                               IF (#statDeviceFaultyModules[#tempSlotIndex + 1] = TRUE)
                               THEN
                                   // Fault in module
                                   #ioSystemData.devices[#tempDeviceIndex].slots[#tempSlotIndex].faulty := TRUE;
                                   #ioSystemData.devices[#tempDeviceIndex].slots[#tempSlotIndex].state := #STATE_FAULT;
                               END_IF;
                           ELSE
                               #ioSystemData.devices[#tempDeviceIndex].slots[#tempSlotIndex].error := FALSE;
                               #ioSystemData.devices[#tempDeviceIndex].slots[#tempSlotIndex].problem := FALSE;
                               #ioSystemData.devices[#tempDeviceIndex].slots[#tempSlotIndex].faulty := FALSE;
                           END_IF;

                           IF (#statDeviceExistingModules[#tempSlotIndex + 1] = TRUE)
                           THEN
                               // Module exists
                               #ioSystemData.devices[#tempDeviceIndex].slots[#tempSlotIndex].exists := TRUE;
                           ELSE
                               // Module does not exist
                               #ioSystemData.devices[#tempDeviceIndex].slots[#tempSlotIndex].exists := FALSE;
                           END_IF;
                       END_IF;
                   END_FOR;
               ELSE
                   // All modules are okay
                   FOR #tempSlotIndex := 0 TO "USERDIAG_SLOTS_PER_DEVICE_UPPER_LIM" DO
                       IF (#ioSystemData.devices[#tempDeviceIndex].slots[#tempSlotIndex].configured = TRUE)
                       THEN
                           #ioSystemData.devices[#tempDeviceIndex].slots[#tempSlotIndex].error := FALSE;
                           #ioSystemData.devices[#tempDeviceIndex].slots[#tempSlotIndex].problem := FALSE;
                           #ioSystemData.devices[#tempDeviceIndex].slots[#tempSlotIndex].faulty := FALSE;
                           #ioSystemData.devices[#tempDeviceIndex].slots[#tempSlotIndex].exists := TRUE;
                       END_IF;
                   END_FOR;
           END_CASE;
       END_IF;

       // Initialize the pointer for the next run
       #tempDeviceIndex := #ioSystemData.devices[#tempDeviceIndex].nextDevice;
   END_WHILE;


   // Write static values to outputs
   #error := #statError;
   #status := #statStatus;
   #statusID := #statStatusID;
END_FUNCTION_BLOCK

FUNCTION_BLOCK "HMI: Network Health"   // FB31, SCL
{ S7_Optimized_Access := 'TRUE' }
VERSION : 0.1
   VAR_IN_OUT
      ioSystemData : Array[1.."USERDIAG_IO_SYSTEMS_UPPER_LIM"] of "UserDiag_typeIOSystem";
      netHealthScreen : "Network Health Screen";
   END_VAR
   VAR_TEMP
      i : Int;
      animate : Struct
         ok : USInt;
         faulty : USInt;
         lostConn : USInt;
         disabled : USInt;
         problem : USInt;
         wasFaulty : USInt;
         wasLost : USInt;
         wasDisabled : USInt;
         problemGone : USInt;
      END_STRUCT;
   END_VAR
   VAR CONSTANT
      statOk : USInt := 1;
   END_VAR
BEGIN
   #animate.ok := "BgDGr";

   FOR #i := 1 TO "pnioDeviceCount" DO
       #netHealthScreen.pnioDevices[#i].label := #ioSystemData[1].devices[#i].name;
       CASE #ioSystemData[1].devices[#i].state OF
           #statOk:
               #netHealthScreen.pnioDevices[#i].animate := #animate.ok;
           ELSE 
               ;
       END_CASE;
   END_FOR;
END_FUNCTION_BLOCK

FUNCTION_BLOCK "HSS: Driver"   // FB32, LAD
{ S7_Optimized_Access := 'TRUE' }
VERSION : 0.1
   VAR_INPUT
      mLs : "Recipe: Libraries";
   END_VAR
   VAR_IN_OUT
      stations : "Stations";
      hmis : Array[0.."hmiStnCount"] of "HSS: Compressed";
   END_VAR
   VAR
      recipeSelector : Array[0.."hmiStnCount"] of Int;
      r1 : Array[0.."hmiStnCount"] of DInt;
      instsHSSMenuSelect : Array[0.."hmiStnCount"] of "HSS: Recipe Selection";
      instsHSSPartSelect : Array[0.."hmiStnCount"] of "HSS: Part Selection";
   END_VAR
   VAR_TEMP
      i : Int;
   END_VAR
   VAR CONSTANT
      hssOffset : Int := 25;
   END_VAR
BEGIN

REGION Network 1 (SCL): TEMPLATE SCREENS
   FOR #i := 0 TO "hmiStnCount" DO
       "HSS: Template"(menuLibrary := #mLs.stations[#i + #hssOffset],
                       menuSelector := #recipeSelector[#i],
                       tmplt := #hmis[#i].scrnTmplt);
       #instsHSSMenuSelect[#i](lib := #mLs.stations[#i + #hssOffset],
                               slctScreen := #hmis[#i].scrnSlctMn,
                               r1 := #r1[#i],
                               station := #stations.me[#i + #hssOffset],
                               recipeSelector := #recipeSelector[#i]);
       #instsHSSPartSelect[#i](recipeNum:= #recipeSelector[#i],
                              lib:=#mLs.stations[#i + #hssOffset],
                              slctScreen:=#hmis[#i].scrnSlctPrt,
                              station:=#stations.me[#i + #hssOffset]);

   END_FOR;
END_REGION
END_FUNCTION_BLOCK

FUNCTION_BLOCK "HSS: Part Selection"   // FB33, SCL
{ S7_Optimized_Access := 'TRUE' }
VERSION : 0.1
   VAR_INPUT
      recipeNum : Int;
      lib : "Recipe: Library";
   END_VAR
   VAR_IN_OUT
      slctScreen : "HSS: Part Selection Screen";
      station : "Station";
   END_VAR
   VAR
      oldBtnsIn : Array[0..31] of Bool;
   END_VAR
   VAR_TEMP
      eval : "HSS: Part Selection Screen";
      i : Int;
      btnsIn : Array[0..31] of Bool;
      btnStates : Array[0.."ptsPerStn"] of Bool;
   END_VAR
BEGIN
   #eval := #slctScreen;


   SCATTER(IN := #slctScreen.pbs ,
           OUT => #btnsIn);
   #btnStates := #station.btnStates;


   FOR #i := 0 TO "ptsPerStn" DO
       IF #btnsIn[#i] AND #btnsIn[#i] <> #oldBtnsIn[#i] THEN
           #btnStates[#i] := NOT #btnStates[#i];
       END_IF;
   END_FOR;


   FOR #i := 0 TO "ptsPerStn" DO
       "Part Select Button"(recipeNum := #recipeNum,
                            lib := #lib,
                            actuate := #btnsIn[#i],
                            btnNum := #i,
                            stn:= #station,
                            partSelectScreen := #eval);
   END_FOR;


   #station.btnStates := #btnStates;
   #oldBtnsIn := #btnsIn;
   #slctScreen := #eval;
END_FUNCTION_BLOCK

FUNCTION_BLOCK "Table Navigatio"   // FB34, SCL
{ S7_Optimized_Access := 'TRUE' }
VERSION : 0.1
   VAR_INPUT
      maxRows : DInt;
      visRows : DInt;
      offset : DInt;
      trigger : Bool;
   END_VAR
   VAR_IN_OUT
      r1 : DInt;
      rowIndices : Array[0..#maxOutRows] of DInt;
   END_VAR
   VAR
      old : Struct
         trigger : Bool := false;
      END_STRUCT;
   END_VAR
   VAR_TEMP
      i : DInt;
      output : Array[0..#maxOutRows] of DInt;
      thisIndex : DInt;
      newR1 : DInt;
   END_VAR
   VAR CONSTANT
      maxOutRows : DInt := 99;
   END_VAR
BEGIN
   IF #trigger AND NOT #old.trigger THEN

       FOR #i := 0 TO #maxOutRows DO
           #output[#i] := -1;
       END_FOR;

       IF #offset > -1000 THEN

           #newR1 := #r1 + #offset;

           IF #newR1 < 0 THEN
               #newR1 := #newR1 + #maxRows;
           END_IF;

           IF #newR1 > #maxRows THEN
               #newR1 := #newR1 - #maxRows;
           END_IF;

       END_IF;

       IF #offset = -1000 THEN
           #newR1 := 0;
       END_IF;

       IF #offset = - 2000 THEN
           #newR1 := #maxRows - #visRows;
       END_IF;

       FOR #i := 0 TO #visRows - 1 DO
           #thisIndex := #newR1 + #i;
           IF #thisIndex < 0 THEN
               #thisIndex := #thisIndex + #maxRows;
           END_IF;
           IF #thisIndex >= #maxRows THEN
               #thisIndex := #thisIndex - #maxRows;
           END_IF;
           #output[#i] := #thisIndex;
       END_FOR;

       #rowIndices := #output;
       #r1 := #newR1;

   END_IF;

   #old.trigger := #trigger;
END_FUNCTION_BLOCK

FUNCTION_BLOCK "HSS: Recipe Selection"   // FB35, SCL
{ S7_Optimized_Access := 'TRUE' }
VERSION : 0.1
   VAR_INPUT
      lib : "Recipe: Library";
   END_VAR
   VAR_IN_OUT
      slctScreen : "HSS: Menu Selection Screen";
      r1 : DInt;
      recipeSelector : Int;
      station : "Station";
   END_VAR
   VAR
      old : Struct
         navPress : Bool;
      END_STRUCT;
      instTableNavigation : "Table Navigatio";
   END_VAR
   VAR_TEMP
      eval : "HSS: Menu Selection Screen";
      pbs : Array[0..#pbFlagCnt] of Bool;
      POS : DInt;
      status : DInt;
      i : Int;
      btnNum : Int;
      pRowVisLbl : Int;
      pRowInvisLbl : Int;
      pRecipeInvisLbl : Int;
      pRecipeVisLbl : Int;
      pRecipeLib : Int;
      pRowTxt : Int;
      pRecipeTxt : Int;
      shifter : DWord;
      btnsAsBool : Array[0..31] of Bool;
      rows : Array[0..99] of DInt;
      offset : DInt;
      navPress : Bool;
      selPress : Bool;
      maxRows : DInt;
      tmrReal : Real;
      partNumber : WString;
   END_VAR
   VAR CONSTANT
      pbFlagCnt : Int := 31;
      btnCnt : Int := 5;
      navMask : DWord := 16#0000_003F;
      visRows : DInt := 6;
      home : DInt := -1000;
      end : DInt := -2000;
      alotted : Real := 1800.0;
      critical : Real := 300.0;
   END_VAR
BEGIN
   REGION "INITITALIZE LOCALS"
       #eval := #slctScreen;
       #maxRows := #lib.size;
       SCATTER(IN := #eval.pbs,
               OUT => #btnsAsBool);
   END_REGION


   REGION "GET RECIPE SELECTION PRESS" 
       FOR #i := 6 TO 31 DO
           IF #btnsAsBool[#i] THEN
               #recipeSelector := DINT_TO_INT(#r1) + #i - 6;
               #selPress := TRUE;
               EXIT;
           END_IF;
       END_FOR;
       FOR #i := 0 TO "ptsPerStn" DO
           #station.partNumbers[#i] := #lib.raw[#recipeSelector, #i];
           // IF #i = 1 THEN
           //     #station.partNumbers[#i] := WSTRING#'';
           // END_IF;

       END_FOR;
       REGION "LOOP THROUGH BUTTONS"
           FOR #i := 0 TO "ptsPerStn" DO

               REGION "COPY TO LOCAL"
                   #partNumber := #station.partNumbers[#i];
               END_REGION

               REGION "IF BUTTON HAS ASSOCIATED PN"
                   IF LEN(#partNumber) <> 0 THEN

                       REGION "COPY TO LOCAL"
                           #tmrReal := #station.presetTime.allotted[#i];
                       END_REGION

                       REGION "ON NO TIME ENTERED"
                           IF #tmrReal = 0.0 THEN

                               REGION "ASSIGN ALLOTTED VALUES"
                                   #station.presetTime.allotted[#i] := #alotted;
                               END_REGION

                           END_IF;
                       END_REGION

                       REGION "COPY TO LOCAL"
                           #tmrReal := #station.presetTime.critical[#i];
                       END_REGION

                       REGION "ON NO TIME ENTERED"
                           IF #tmrReal = 0.0 THEN

                               REGION "ASSIGN CRITICAL VALUES"
                                   #station.presetTime.critical[#i] := #critical;
                               END_REGION

                           END_IF;
                       END_REGION

                   END_IF;
               END_REGION

               REGION "IF BUTTON HAS NO ASSOCIATED PN"
                   IF LEN(#partNumber) = 0 THEN

                       REGION "COPY TO LOCAL"
                           #tmrReal := #station.presetTime.allotted[#i];
                       END_REGION

                       REGION "ON NO TIME ENTERED"
                           IF #tmrReal <> 0.0 THEN

                               REGION "ASSIGN ALLOTTED VALUES"
                                   #station.presetTime.allotted[#i] := 0.0;
                               END_REGION

                           END_IF;
                       END_REGION

                       REGION "COPY TO LOCAL"
                           #tmrReal := #station.presetTime.critical[#i];
                       END_REGION

                       REGION "ON NO TIME ENTERED"
                           IF #tmrReal <> 0.0 THEN

                               REGION "ASSIGN CRITICAL VALUES"
                                   #station.presetTime.critical[#i] := 0.0;
                               END_REGION

                           END_IF;
                       END_REGION

                   END_IF;
               END_REGION


           END_FOR;
       END_REGION
   END_REGION


   REGION "TABLE NAVIGATION"
       IF #maxRows > #visRows THEN
           IF #eval.pbs.%X0 THEN
               #offset := #home;
           END_IF;
           IF #eval.pbs.%X1 THEN
               #offset := -1 * #visRows;
           END_IF;
           IF #eval.pbs.%X2 THEN
               #offset := -1;
           END_IF;
           IF #eval.pbs.%X3 THEN
               #offset := 1;
           END_IF;
           IF #eval.pbs.%X4 THEN
               #offset := #visRows;
           END_IF;
           IF #eval.pbs.%X5 THEN
               #offset := #end;
           END_IF;

           IF (#eval.pbs AND #navMask) <> 0 THEN
               #navPress := true;
           END_IF;

           #instTableNavigation(maxRows := #maxRows,
                                visRows := #visRows,
                                offset := #offset,
                                trigger := #navPress,
                                r1 := #r1,
                                rowIndices := #rows);
       END_IF;

       IF #maxRows <= #visRows THEN
           FOR #i := 0 TO #visRows - 1 DO
               #rows[#i] := #i;
           END_FOR;
       END_IF;

   END_REGION


   REGION "CA: NAV BUTTONS"
       FOR #i := 0 TO #visRows - 1 DO
           "Recipe Nav Button"(visRows := DINT_TO_INT(#visRows),
                               actuate := #btnsAsBool[#i],
                               maxRows := DINT_TO_INT(#maxRows),
                               btnNum := #i,
                               recipeSelectScreen := #eval);
       END_FOR;
   END_REGION



   REGION "ODA: RECIPE SELECT BUTTONS"
       IF (#navPress AND NOT #old.navPress) OR
           (#maxRows <= #visRows) THEN

           FOR #i := 0 TO #visRows - 1 DO
               "Recipe Select Button"(visRows := DINT_TO_INT(#visRows),
                                      rowNum := DINT_TO_INT(#rows[#i]),
                                      lib := #lib,
                                      actuate := #btnsAsBool[#i + 6],
                                      maxRows := DINT_TO_INT(#maxRows),
                                      btnNum := #i,
                                      recipeSelectScreen := #eval);
           END_FOR;

       END_IF;
   END_REGION


   REGION "CHANGE DETECTION"
       #old.navPress := #navPress;
   END_REGION


   REGION "COPY TO GLOBAL"
       #slctScreen := #eval;
   END_REGION
END_FUNCTION_BLOCK

FUNCTION_BLOCK "KP8 Driver"   // FB101, SCL
{ S7_Optimized_Access := 'FALSE' }
VERSION : 0.1
   VAR_INPUT
      btnIn : Byte;   // byte that contains input data from kp8 buttons
      hardInit : Bool;   // initializes function. can be used for reset
      softInit : Bool;
      btn0Activate : Bool;   // true for on, false for off
      btn0Mode : Bool;   // true for maintained, false for momentary
      btn0Group : Int;
      btn0Flash : Bool;
      btn0ColorOn1 : String[10];   // enter: red OR green OR blue OR yellow OR white OR off
      btn0ColorOn2 : String[10];
      btn0ColorOff : String[10];   // enter: red OR green OR blue OR yellow OR white OR off
      btn1Activate : Bool;   // true for on, false for off
      btn1Mode : Bool;   // true for maintained, false for momentary
      btn1Group : Int;
      btn1Flash : Bool;
      btn1ColorOn1 : String[10];   // enter: red OR green OR blue OR yellow OR white OR off
      btn1ColorOn2 : String[10];
      btn1ColorOff : String[10];   // enter: red OR green OR blue OR yellow OR white OR off
      btn2Activate : Bool;   // true for on, false for off
      btn2Mode : Bool;   // true for maintained, false for momentary
      btn2Group : Int;
      btn2Flash : Bool;
      btn2ColorOn1 : String[10] := '';   // enter: red OR green OR blue OR yellow OR white OR off
      btn2ColorOn2 : String[10];
      btn2ColorOff : String[10];   // enter: red OR green OR blue OR yellow OR white OR off
      btn3Activate : Bool;   // true for on, false for off
      btn3Mode : Bool;   // true for maintained, false for momentary
      btn3Group : Int;
      btn3Flash : Bool;
      btn3ColorOn1 : String[10];   // enter: red OR green OR blue OR yellow OR white OR off
      btn3ColorOn2 : String[10];
      btn3ColorOff : String[10];   // enter: red OR green OR blue OR yellow OR white OR off
      btn4Activate : Bool;   // true for on, false for off
      btn4Mode : Bool;   // true for maintained, false for momentary
      btn4Group : Int;
      btn4Flash : Bool;
      btn4ColorOn1 : String[10];   // enter: red OR green OR blue OR yellow OR white OR off
      btn4ColorOn2 : String[10];
      btn4ColorOff : String[10];   // enter: red OR green OR blue OR yellow OR white OR off
      btn5Activate : Bool;   // true for on, false for off
      btn5Mode : Bool;   // true for maintained, false for momentary
      btn5Group : Int;
      btn5Flash : Bool;
      btn5ColorOn1 : String[10];   // enter: red OR green OR blue OR yellow OR white OR off
      btn5ColorOn2 : String[10];
      btn5ColorOff : String[10];   // enter: red OR green OR blue OR yellow OR white OR off
      btn6Activate : Bool;   // true for on, false for off
      btn6Mode : Bool;   // true for maintained, false for momentary
      btn6Group : Int;
      btn6Flash : Bool;
      btn6ColorOn1 : String[10];   // enter: red OR green OR blue OR yellow OR white OR off
      btn6ColorOn2 : String[10];
      btn6ColorOff : String[10];   // enter: red OR green OR blue OR yellow OR white OR off
      btn7Activate : Bool;   // true for on, false for off
      btn7Mode : Bool;   // true for maintained, false for momentary
      btn7Group : Int;
      btn7Flash : Bool;
      btn7ColorOn1 : String[10];   // enter: red OR green OR blue OR yellow OR white OR off
      btn7ColorOn2 : String[10];
      btn7ColorOff : String[10];   // enter: red OR green OR blue OR yellow OR white OR off
   END_VAR
   VAR_OUTPUT
      btnStatesOut : Array[0..7] of Bool;   // the output array represents the state of button presses
      btnColorsOut : DWord;
   END_VAR
   VAR
      mask : Byte;
      btnInInt : Byte;
      btnEval : Byte;
      i1 : Int;
      i2 : Int;
      btnActivateInt : Array[0..7] of Bool;
      btnClrMskOffInt : Array[0..7] of DWord;
      btnClrMskOn1Int : Array[0..7] of DWord;
      btnClrMskOn2Int : Array[0..7] of DWord;
      btnClrOffInt : Array[0..7] of String[10];
      btnClrOn1Int : Array[0..7] of String[10];
      btnClrOn2Int : Array[0..7] of String[10];
      btnColors : DWord;
      btnInArrayNew : Array[0..7] of Bool;
      btnInArrayOld : Array[0..7] of Bool;
      btnStateArrayInt : Array[0..7] of Bool;
      btnModeInt : Array[0..7] of Bool;
      btnFlashInt : Array[0..7] of Bool;
      btnGroup : Array[0..7] of Int;
   END_VAR
   VAR CONSTANT
      btnMskRed : DWord := dw#16#0100_0000;
      btnMskGreen : DWord := dw#16#0001_0000;
      btnMskBlue : DWord := dw#16#000_0100;
      btnMskYellow : DWord := dw#16#0101_0000;
      btnMskWhite : DWord := dw#16#0101_0100;
      btnMskBlack : DWord := dw#16#FEFE_FEFF;
      initBtnColors : DWord := dw#16#0000_0000;
   END_VAR
BEGIN
   REGION "ALL INITS"
       IF #hardInit OR #softInit THEN

           REGION "CLEAR OUTPUT COLORS"
               #btnColors := #initBtnColors;
           END_REGION

           REGION "TRANSFER PARAMETERS TO INTERNAL ARRAYS"

               REGION "BUTTON 0"
                   #btnActivateInt[0] := #btn0Activate;
                   #btnModeInt[0] := #btn0Mode;
                   #btnGroup[0] := #btn0Group;
                   #btnClrOn1Int[0] := #btn0ColorOn1;
                   #btnClrOn2Int[0] := #btn0ColorOn2;
                   #btnClrOffInt[0] := #btn0ColorOff;
               END_REGION

               REGION "BUTTON 1"
                   #btnActivateInt[1] := #btn1Activate;
                   #btnModeInt[1] := #btn1Mode;
                   #btnGroup[1] := #btn1Group;
                   #btnClrOn1Int[1] := #btn1ColorOn1;
                   #btnClrOn2Int[1] := #btn1ColorOn2;
                   #btnClrOffInt[1] := #btn1ColorOff;
               END_REGION

               REGION "BUTTON 2"
                   #btnActivateInt[2] := #btn2Activate;
                   #btnModeInt[2] := #btn2Mode;
                   #btnGroup[2] := #btn2Group;
                   #btnClrOn1Int[2] := #btn2ColorOn1;
                   #btnClrOn2Int[2] := #btn2ColorOn2;
                   #btnClrOffInt[2] := #btn2ColorOff;
               END_REGION

               REGION "BUTTON 3"
                   #btnActivateInt[3] := #btn3Activate;
                   #btnModeInt[3] := #btn3Mode;
                   #btnGroup[3] := #btn3Group;
                   #btnClrOn1Int[3] := #btn3ColorOn1;
                   #btnClrOn2Int[3] := #btn3ColorOn2;
                   #btnClrOffInt[3] := #btn3ColorOff;
               END_REGION

               REGION "BUTTON 4"
                   #btnActivateInt[4] := #btn4Activate;
                   #btnModeInt[4] := #btn4Mode;
                   #btnGroup[4] := #btn4Group;
                   #btnClrOn1Int[4] := #btn4ColorOn1;
                   #btnClrOn2Int[4] := #btn4ColorOn2;
                   #btnClrOffInt[4] := #btn4ColorOff;
               END_REGION

               REGION "BUTTON 5"
                   #btnActivateInt[5] := #btn5Activate;
                   #btnModeInt[5] := #btn5Mode;
                   #btnGroup[5] := #btn5Group;
                   #btnClrOn1Int[5] := #btn5ColorOn1;
                   #btnClrOn2Int[5] := #btn5ColorOn2;
                   #btnClrOffInt[5] := #btn5ColorOff;
               END_REGION

               REGION "BUTTON 6"
                   #btnActivateInt[6] := #btn6Activate;
                   #btnModeInt[6] := #btn6Mode;
                   #btnGroup[6] := #btn6Group;
                   #btnClrOn1Int[6] := #btn6ColorOn1;
                   #btnClrOn2Int[6] := #btn6ColorOn2;
                   #btnClrOffInt[6] := #btn6ColorOff;
               END_REGION

               REGION "BUTTON 7"
                   #btnActivateInt[7] := #btn7Activate;
                   #btnModeInt[7] := #btn7Mode;
                   #btnGroup[7] := #btn7Group;
                   #btnClrOn1Int[7] := #btn7ColorOn1;
                   #btnClrOn2Int[7] := #btn7ColorOn2;
                   #btnClrOffInt[7] := #btn7ColorOff;
               END_REGION

           END_REGION

           REGION "RECOLOR BUTTON MASKS"
               FOR #i1 := 0 TO 7 DO

                   REGION "ON COLOR 1"
                       IF (#btnClrOn1Int[#i1] = 'red') THEN
                           #btnClrMskOn1Int[#i1] := SHL(IN := #btnMskRed, N := INT_TO_ULINT(#i1));
                       ELSIF (#btnClrOn1Int[#i1] = 'green') THEN
                           #btnClrMskOn1Int[#i1] := SHL(IN := #btnMskGreen, N := INT_TO_ULINT(#i1));
                       ELSIF (#btnClrOn1Int[#i1] = 'blue') THEN
                           #btnClrMskOn1Int[#i1] := SHL(IN := #btnMskBlue, N := INT_TO_ULINT(#i1));
                       ELSIF (#btnClrOn1Int[#i1] = 'yellow') THEN
                           #btnClrMskOn1Int[#i1] := SHL(IN := #btnMskYellow, N := INT_TO_ULINT(#i1));
                       ELSIF (#btnClrOn1Int[#i1] = 'white') THEN
                           #btnClrMskOn1Int[#i1] := SHL(IN := #btnMskWhite, N := INT_TO_ULINT(#i1));
                       ELSIF (#btnClrOn1Int[#i1] = 'off') THEN
                           #btnClrMskOn1Int[#i1] := 0;
                       END_IF;
                   END_REGION

                   REGION "ON COLOR 2"
                       IF (#btnClrOn2Int[#i1] = 'red') THEN
                           #btnClrMskOn2Int[#i1] := SHL(IN := #btnMskRed, N := INT_TO_ULINT(#i1));
                       ELSIF (#btnClrOn2Int[#i1] = 'green') THEN
                           #btnClrMskOn2Int[#i1] := SHL(IN := #btnMskGreen, N := INT_TO_ULINT(#i1));
                       ELSIF (#btnClrOn2Int[#i1] = 'blue') THEN
                           #btnClrMskOn2Int[#i1] := SHL(IN := #btnMskBlue, N := INT_TO_ULINT(#i1));
                       ELSIF (#btnClrOn2Int[#i1] = 'yellow') THEN
                           #btnClrMskOn2Int[#i1] := SHL(IN := #btnMskYellow, N := INT_TO_ULINT(#i1));
                       ELSIF (#btnClrOn2Int[#i1] = 'white') THEN
                           #btnClrMskOn2Int[#i1] := SHL(IN := #btnMskWhite, N := INT_TO_ULINT(#i1));
                       ELSIF (#btnClrOn2Int[#i1] = 'off') THEN
                           #btnClrMskOn2Int[#i1] := 0;
                       END_IF;
                   END_REGION

                   REGION "OFF COLOR"
                       IF (#btnClrOffInt[#i1] = 'red') THEN
                           #btnClrMskOffInt[#i1] := SHL(IN := #btnMskRed, N := INT_TO_ULINT(#i1));
                       ELSIF (#btnClrOffInt[#i1] = 'green') THEN
                           #btnClrMskOffInt[#i1] := SHL(IN := #btnMskGreen, N := INT_TO_ULINT(#i1));
                       ELSIF (#btnClrOffInt[#i1] = 'blue') THEN
                           #btnClrMskOffInt[#i1] := SHL(IN := #btnMskBlue, N := INT_TO_ULINT(#i1));
                       ELSIF (#btnClrOffInt[#i1] = 'yellow') THEN
                           #btnClrMskOffInt[#i1] := SHL(IN := #btnMskYellow, N := INT_TO_ULINT(#i1));
                       ELSIF (#btnClrOffInt[#i1] = 'white') THEN
                           #btnClrMskOffInt[#i1] := SHL(IN := #btnMskWhite, N := INT_TO_ULINT(#i1));
                       ELSIF (#btnClrOffInt[#i1] = 'off') THEN
                           #btnClrMskOffInt[#i1] := 0;
                       END_IF;
                   END_REGION

               END_FOR;
           END_REGION

       END_IF;
   END_REGION

   REGION "HART INIT"
       IF #hardInit THEN
           FOR #i1 := 0 TO 7 DO
               #btnStateArrayInt[#i1] := FALSE;
           END_FOR;
       END_IF;
   END_REGION


   REGION "TRANFER PARAMETERS TO ARRAYS"
       // raw pb data
       #btnInInt := #btnIn;
       // flashing modes
       #btnFlashInt[0] := #btn0Flash;
       #btnFlashInt[1] := #btn1Flash;
       #btnFlashInt[2] := #btn2Flash;
       #btnFlashInt[3] := #btn3Flash;
       #btnFlashInt[4] := #btn4Flash;
       #btnFlashInt[5] := #btn5Flash;
       #btnFlashInt[6] := #btn6Flash;
       #btnFlashInt[7] := #btn7Flash;
   END_REGION

   REGION "EVALUATE BUTTONS"
       FOR #i1 := 0 TO 7 DO

           REGION "TRANSFER BUTTON PRESSES TO ARRAY"
               #btnEval := SHR(IN := #btnInInt, N := INT_TO_ULINT(#i1));
               #btnInArrayNew[#i1] := #btnEval.%X0;
               #btnEval := b#16#0;
           END_REGION

           REGION "SET BUTTON STATE"

               REGION "BUTTON ACTIVE"
                   IF #btnActivateInt[#i1] THEN

                       REGION "MAINTAINED"
                           IF #btnModeInt[#i1] THEN

                               REGION "RISING EDGE OF PRESS"
                                   IF #btnInArrayNew[#i1] AND NOT #btnInArrayOld[#i1] THEN

                                       REGION "CHECK FOR GROUP MEMBERSHIP"
                                           FOR #i2 := 0 TO 7 DO

                                               REGION "NOT IN NULL GROUP"
                                                   IF (#btnGroup[#i2] <> 0) THEN

                                                       REGION "SKIP SELF"
                                                           IF (#i2 <> #i1) THEN

                                                               REGION "GROUPS MATCH"
                                                                   IF #btnGroup[#i1] = #btnGroup[#i2] THEN
                                                                       REGION "DEACTIVATE OTHER GROUP MEMBERS"
                                                                           #btnStateArrayInt[#i2] := FALSE;
                                                                       END_REGION

                                                                   END_IF;
                                                               END_REGION

                                                           END_IF;
                                                       END_REGION

                                                   END_IF;
                                               END_REGION

                                           END_FOR;
                                       END_REGION

                                       REGION "TOGGLE STATE"
                                           #btnStateArrayInt[#i1] := NOT #btnStateArrayInt[#i1];
                                       END_REGION

                                   END_IF;
                               END_REGION

                           END_IF;
                       END_REGION

                       REGION "MOMENTARY"
                           IF NOT #btnModeInt[#i1] THEN
                               #btnStateArrayInt[#i1] := #btnInArrayNew[#i1];
                           END_IF;
                       END_REGION

                   END_IF;
               END_REGION

               REGION "BUTTON INACTIVE"
                   IF NOT #btnActivateInt[#i1] THEN
                       #btnStateArrayInt[#i1] := FALSE;
                   END_IF;
               END_REGION

           END_REGION

           REGION "ANIMATE BUTTONS"

               REGION "BUTTON ON FLASH BIT OFF"
                   IF #btnStateArrayInt[#i1] AND NOT #btnFlashInt[#i1] THEN
                       #btnColors := #btnColors AND ROL(IN := #btnMskBlack, N := INT_TO_ULINT(#i1));
                       #btnColors := #btnColors OR #btnClrMskOn1Int[#i1];
                   END_IF;
               END_REGION

               REGION "BUTTON ON FLASH BIT ON"
                   IF #btnStateArrayInt[#i1] AND #btnFlashInt[#i1] THEN
                       #btnColors := #btnColors AND ROL(IN := #btnMskBlack, N := INT_TO_ULINT(#i1));
                       #btnColors := #btnColors OR #btnClrMskOn2Int[#i1];
                   END_IF;
               END_REGION

               REGION "BUTTON OFF"
                   IF NOT #btnStateArrayInt[#i1] THEN
                       #btnColors := #btnColors AND ROL(IN := #btnMskBlack, N := INT_TO_ULINT(#i1));
                       #btnColors := #btnColors OR #btnClrMskOffInt[#i1];
                   END_IF;
               END_REGION

           END_REGION

       END_FOR;
   END_REGION

   REGION "CHANGE DETECTION"
       #btnInArrayOld := #btnInArrayNew;
   END_REGION

   REGION "OUTPUT"
       #btnColorsOut := #btnColors;
       #btnStatesOut := #btnStateArrayInt;
   END_REGION
END_FUNCTION_BLOCK

FUNCTION "Physical to Global" : Void   // FC1, LAD
{ S7_Optimized_Access := 'TRUE' }
VERSION : 0.1
   VAR_IN_OUT
      stations : "Stations";
   END_VAR
   VAR_TEMP
      i : Int;
      kp8In : DWord;
   END_VAR
BEGIN

REGION Network 1 (SCL): MAIN LOOP
   FOR #i := 0 TO "stnCount" DO

       CASE #i OF
           "VOLVO 16 01":
               #kp8In := "VOLVO 16 01 KP8 In";
           "VOLVO 16 02":
               #kp8In := "VOLVO 16 02 KP8 In";
           "VOLVO 16 03":
               #kp8In := "VOLVO 16 03 KP8 In";
           "VOLVO 16 04":
               #kp8In := "VOLVO 16 04 KP8 In";
           "VOLVO 16 05":
               #kp8In := "VOLVO 16 05 KP8 In";
           "VOLVO 16 06":
               #kp8In := "VOLVO 16 06 KP8 In";
           "VOLVO 16 07":
               #kp8In := "VOLVO 16 07 KP8 In";
           "VOLVO 16 08":
               #kp8In := "VOLVO 16 08 KP8 In";
           "VOLVO 16 09":
               #kp8In := "VOLVO 16 09 KP8 In";
           "VOLVO 16 10":
               #kp8In := "VOLVO 16 10 KP8 In";
           "VOLVO 16 11":
               #kp8In := "VOLVO 16 11 KP8 In";
           "CHM 01":
               #kp8In := "CHM 01 KP8 In";
           "CHM 02":
               #kp8In := "CHM 02 KP8 In";
           "CHM 03":
               #kp8In := "CHM 03 KP8 In";
           "CHM 04":
               #kp8In := "CHM 04 KP8 In";
           "CHM 05":
               #kp8In := "CHM 05 KP8 In";
           "CDO 01":
               #kp8In := "CDO 01 KP8 In";
           "CDO 02":
               #kp8In := "CDO 02 KP8 In";
           "CDO 03":
               #kp8In := "CDO 03 KP8 In";
           "BFL 01":
               #kp8In := "BFL 01 KP8 In";
           "BFL 02":
               #kp8In := "BFL 02 KP8 In";
           "BFL 03":
               #kp8In := "BFL 03 KP8 In";
           "LGS 01":
               #kp8In := "LGS 01 KP8 In";
           "LGS 02":
               #kp8In := "LGS 02 KP8 In";
           "LGS 03":
               #kp8In := "LGS 03 KP8 In";
           "CV 01":
               #kp8In := "CV 01 KP8 In";
           "CV 02":
               #kp8In := "CV 02 KP8 In";
           "CV 03":
               #kp8In := "CV 03 KP8 In";
           "CV 04":
               #kp8In := "CV 04 KP8 In";
           "PC 01":
               #kp8In := "PC 01 KP8 In"; 
           "PC 02":
               #kp8In := "PC 02 KP8 In";
           "1BX 2.0 01":
               #kp8In := "1BX 2.0 01 KP8 In";
           "1BX 2.0 02":
               #kp8In := "1BX 2.0 02 KP8 In";
           "1BX 2.0 03":
               #kp8In := "1BX 2.0 03 KP8 In";
           "1BX 2.0 04":
               #kp8In := "1BX 2.0 04 KP8 In";
           "1BX 2.0 05":
               #kp8In := "1BX 2.0 05 KP8 In";
           "1BX 3.0 01":
               #kp8In := "1BX 3.0 01 KP8 In";
           "1BX 3.0 02":
               #kp8In := "1BX 3.0 02 KP8 In";
           "1BX 3.0 03":
               #kp8In := "1BX 3.0 03 KP8 In";


       END_CASE;

       #stations.me[#i].kp8In := #kp8In.%B3;

   END_FOR;
END_REGION
END_FUNCTION

FUNCTION "Time to WString" : WString   // FC2, SCL
{ S7_Optimized_Access := 'TRUE' }
VERSION : 0.1
   VAR_INPUT
      "Time" : Time;
   END_VAR
   VAR_TEMP
      "Time as DInt" : DInt;
      "Hours 10s Place" : DInt;
      "Hours 1s Place" : DInt;
      "Minutes 10s Place" : DInt;
      "Minutes 1s Place" : DInt;
      "Seconds 10s Place" : DInt;
      "Seconds 1s Place" : DInt;
      "Time Elements" : Array[0..4] of WString;
      Length : Int;
      "String Box" : WString;
      "DInt Box" : DInt;
   END_VAR
   VAR CONSTANT
      "Milliseconds per 10 Hours" : DInt := 36000000;
      "Milliseconds per Hour" : DInt := 3600000;
      "Milliseconds per 10 Minutes" : DInt := 600000;
      "Milliseconds per Minute" : DInt := 60000;
      "Milliseconds per 10 Seconds" : DInt := 10000;
      "Milliseconds per Second" : DInt := 1000;
   END_VAR
BEGIN
   REGION GET INPUT
       #"Time as DInt" := #Time;
   END_REGION

   REGION CONVERT TIME INTO INDIVIDUAL PLACE VALUES
       #"Minutes 10s Place" := #"Time as DInt" / #"Milliseconds per 10 Minutes";
       #"Minutes 1s Place" := (#"Time as DInt" / #"Milliseconds per Minute") MOD 10;
       #"Seconds 10s Place" := (#"Time as DInt" MOD #"Milliseconds per Minute") / #"Milliseconds per 10 Seconds";
       #"Seconds 1s Place" := (#"Time as DInt" / #"Milliseconds per Second") MOD 10;
   END_REGION

   REGION "ADD SIGN"
       #"Time Elements"[0] := wstring#'';
       IF #"Minutes 10s Place" < 0 OR
           #"Minutes 1s Place" < 0 OR
           #"Seconds 10s Place" < 0 OR
           #"Seconds 1s Place" < 0 THEN
            #"Time Elements"[0] := wstring#'-';
       END_IF;
   END_REGION

   REGION CONVERT PLACE VALUES INTO COMPONENT STRINGS
       // MINUTES
       #"DInt Box" := #"Minutes 10s Place" * 10 + #"Minutes 1s Place";
       #"String Box" := DINT_TO_WSTRING(IN := #"DInt Box");
       #"String Box" := "Strip Sign"("WString":=#"String Box");
       #"String Box" := "Add Leading"("Leading Character" := WCHAR#'0',
                                      "Desired Length" := 2,
                                      "String" := #"String Box");
       #"Time Elements"[1] := #"String Box";
       // COLON
       #"Time Elements"[2] := WSTRING#':';
       // SECONDS
       #"DInt Box" := #"Seconds 10s Place" * 10 + #"Seconds 1s Place";
       #"String Box" := DINT_TO_WSTRING(IN := #"DInt Box");
       #"String Box" := "Strip Sign"("WString":=#"String Box");
       #"String Box" := "Add Leading"("Leading Character" := WCHAR#'0',
                                      "Desired Length" := 2,
                                      "String" := #"String Box");
       #"Time Elements"[3] := #"String Box";
   END_REGION


   REGION RETURN VALUE
       #"Time to WString" := CONCAT_WSTRING(IN1 := #"Time Elements"[0],
                                            IN2 := #"Time Elements"[1],
                                            IN3 := #"Time Elements"[2],
                                            IN4 := #"Time Elements"[3]);
   END_REGION
END_FUNCTION

FUNCTION "Strip Sign" : WString   // FC3, SCL
{ S7_Optimized_Access := 'TRUE' }
VERSION : 0.1
   VAR_INPUT
      WString : WString;
   END_VAR
   VAR_TEMP
      Length : Int;
      "String Box" : WString;
      "Test Character" : WString;
   END_VAR
   VAR CONSTANT
      "+" : WChar := WCHAR#'+';
      "-" : WChar := WCHAR#'-';
   END_VAR
BEGIN
   #"String Box" := #WString;
   #"Test Character" := LEFT_WSTRING(IN := #"String Box",
                                     L := 1);
   IF #"Test Character" = #"+" OR #"Test Character" = #"-" THEN
       #Length := LEN(#"String Box");
       #"String Box" := RIGHT_WSTRING(IN := #"String Box", L := #Length - 1);

   END_IF;
   #"Strip Sign" := #"String Box";
END_FUNCTION

FUNCTION "Add Leading" : WString   // FC4, SCL
{ S7_Optimized_Access := 'TRUE' }
VERSION : 0.1
   VAR_INPUT
      "Leading Character" : WChar;
      "Desired Length" : USInt;
      "String" : WString;
   END_VAR
   VAR_TEMP
      Length : Int;
      "String Box" : WString;
      Constant : WString;
   END_VAR
BEGIN
   #"String Box" := #String;
   #Length := LEN(#"String Box");

   WHILE #Length < #"Desired Length" DO
       #"String Box" := CONCAT_WSTRING(IN1 := #"Leading Character",
                                       IN2 := #"String Box");
       #Length := LEN(#"String Box");
   END_WHILE;

   #"Add Leading" := #"String Box";
END_FUNCTION

FUNCTION "Global to Physical" : Void   // FC5, LAD
{ S7_Optimized_Access := 'TRUE' }
VERSION : 0.1
   VAR_IN_OUT
      stations : "Stations";
   END_VAR
   VAR_TEMP
      i : Int;
      j : Int;
      IO : DWord;
      "KP8 In" : DWord;
      "KP8 Out" : DWord;
      Card : Int;
      stnCount : Int;
   END_VAR
BEGIN

REGION Network 1 (SCL): MAIN LOOP
   FOR #i := 0 TO "stnCount" DO

       #IO := #stations.me[#i].stackLightOut;
       #"KP8 Out" := #stations.me[#i].kp8Out;

       CASE #i OF
           "VOLVO 16 01":
               "VOLVO 16 01 IO" := #IO;
               "VOLVO 16 01 KP8 Out" := #"KP8 Out";
           "VOLVO 16 02":
               "VOLVO 16 02 IO" := #IO;
               "VOLVO 16 02 KP8 Out" := #"KP8 Out";
           "VOLVO 16 03":
               "VOLVO 16 03 IO" := #IO;
               "VOLVO 16 03 KP8 Out" := #"KP8 Out";
           "VOLVO 16 04":
               "VOLVO 16 04 IO" := #IO;
               "VOLVO 16 04 KP8 Out" := #"KP8 Out";
           "VOLVO 16 05":
               "VOLVO 16 05 IO" := #IO;
               "VOLVO 16 05 KP8 Out" := #"KP8 Out";
           "VOLVO 16 06":
               "VOLVO 16 06 IO" := #IO;
               "VOLVO 16 06 KP8 Out" := #"KP8 Out";
           "VOLVO 16 07":
               "VOLVO 16 07 IO" := #IO;
               "VOLVO 16 07 KP8 Out" := #"KP8 Out";
           "VOLVO 16 08":
               "VOLVO 16 08 IO" := #IO;
               "VOLVO 16 08 KP8 Out" := #"KP8 Out";
           "VOLVO 16 09":
               "VOLVO 16 09 IO" := #IO;
               "VOLVO 16 09 KP8 Out" := #"KP8 Out";
           "VOLVO 16 10":
               "VOLVO 16 10 IO" := #IO;
               "VOLVO 16 10 KP8 Out" := #"KP8 Out";
           "VOLVO 16 11":
               "VOLVO 16 11 IO" := #IO;
               "VOLVO 16 11 KP8 Out" := #"KP8 Out";
           "CHM 01":
               "CHM 01 IO" := #IO;
               "CHM 01 KP8 Out" := #"KP8 Out";
           "CHM 02":
               "CHM 02 IO" := #IO;
               "CHM 02 KP8 Out" := #"KP8 Out";
           "CHM 03":
               "CHM 03 IO" := #IO;
               "CHM 03 KP8 Out" := #"KP8 Out";
           "CHM 04":
               "CHM 04 IO" := #IO;
               "CHM 04 KP8 Out" := #"KP8 Out";
           "CHM 05":
               "CHM 05 IO" := #IO;
               "CHM 05 KP8 Out" := #"KP8 Out";
           "CDO 01":
               "CDO 01 IO" := #IO;
               "CDO 01 KP8 Out" := #"KP8 Out";
           "CDO 02":
               "CDO 02 IO" := #IO;
               "CDO 02 KP8 Out" := #"KP8 Out";
           "CDO 03":
               "CDO 03 IO" := #IO;
               "CDO 03 KP8 Out" := #"KP8 Out";
           "BFL 01":
               "BFL 01 IO" := #IO;
               "BFL 01 KP8 Out" := #"KP8 Out";
           "BFL 02":
               "BFL 02 IO" := #IO;
               "BFL 02 KP8 Out" := #"KP8 Out";
           "BFL 03":
               "BFL 03 IO" := #IO;
               "BFL 03 KP8 Out" := #"KP8 Out";
           "LGS 01":
               "LGS 01 IO" := #IO;
               "LGS 01 KP8 Out" := #"KP8 Out";
           "LGS 02":
               "LGS 02 IO" := #IO;
               "LGS 02 KP8 Out" := #"KP8 Out";
           "LGS 03":
               "LGS 03 IO" := #IO;
               "LGS 03 KP8 Out" := #"KP8 Out";
           "CV 01":
               "CV 01 IO" := #IO;
               "CV 01 KP8 Out" := #"KP8 Out";
           "CV 02":
               "CV 02 IO" := #IO;
               "CV 02 KP8 Out" := #"KP8 Out";
           "CV 03":
               "CV 03 IO" := #IO;
               "CV 03 KP8 Out" := #"KP8 Out";
           "CV 04":
               "CV 04 IO" := #IO;
               "CV 04 KP8 Out" := #"KP8 Out";
           "PC 01":
               "PC 01 IO" := #IO;
               "PC 01 KP8 Out" := #"KP8 Out";
           "PC 02":
               "PC 02 IO" := #IO;
               "PC 02 KP8 Out" := #"KP8 Out";
           "1BX 2.0 01":
               "1BX 2.0 01 IO" := #IO;
               "1BX 2.0 01 KP8 Out" := #"KP8 Out";
           "1BX 2.0 02":
               "1BX 2.0 02 IO" := #IO;
               "1BX 2.0 02 KP8 Out" := #"KP8 Out";
           "1BX 2.0 03":
               "1BX 2.0 03 IO" := #IO;
               "1BX 2.0 03 KP8 Out" := #"KP8 Out";
           "1BX 2.0 04":
               "1BX 2.0 04 IO" := #IO;
               "1BX 2.0 04 KP8 Out" := #"KP8 Out";
           "1BX 2.0 05":
               "1BX 2.0 05 IO" := #IO;
               "1BX 2.0 05 KP8 Out" := #"KP8 Out";
           "1BX 3.0 01":
               "1BX 3.0 01 IO" := #IO;
               "1BX 3.0 01 KP8 Out" := #"KP8 Out";
           "1BX 3.0 02":
               "1BX 3.0 02 IO" := #IO;
               "1BX 3.0 02 KP8 Out" := #"KP8 Out";
           "1BX 3.0 03":
               "1BX 3.0 03 IO" := #IO;
               "1BX 3.0 03 KP8 Out" := #"KP8 Out";

       END_CASE;

   END_FOR;
END_REGION
END_FUNCTION

FUNCTION "Select Stations" : Void   // FC6, SCL
{ S7_Optimized_Access := 'TRUE' }
VERSION : 0.1
   VAR_INPUT
      mode : Bool;   // TRUE = select; FALSE = deselect
   END_VAR
   VAR_IN_OUT
      stations : "Stations";
   END_VAR
   VAR_TEMP
      i : Int;
      stnCount : Int;
   END_VAR
   VAR CONSTANT
      stationCount : Int := 22;
   END_VAR
BEGIN
   REGION "GET STATION COUNT"
       #stnCount := "stnCount";
   END_REGION

   REGION "SELECT STATIONS"
       FOR #i := 0 TO #stnCount DO
           #stations.me[#i].settings.selected := #mode;
       END_FOR;
   END_REGION
END_FUNCTION

FUNCTION "Dark Mode" : Void   // FC7, SCL
{ S7_Optimized_Access := 'TRUE' }
VERSION : 0.1
   VAR_IN_OUT
      animate : USInt;
   END_VAR
   VAR_TEMP
      ani : USInt;
   END_VAR
   VAR CONSTANT
      redFlashing : USInt := 12;
      invisible : USInt := 255;
      darkMode : USInt := 1;
      disabled : USInt := 254;
   END_VAR
BEGIN
   REGION "COPY TO LOCAL"
       #ani := #animate;
   END_REGION


   REGION "APPLY DARK MODE"
       CASE #ani OF
           #redFlashing, #invisible, 0, #disabled:
               #ani := #ani;
           ELSE
               #ani += #darkMode;
       END_CASE;
   END_REGION


   REGION "OUTPUT"
       #animate := #ani;
   END_REGION
END_FUNCTION

FUNCTION "Select Buttons" : Void   // FC8, SCL
{ S7_Optimized_Access := 'TRUE' }
VERSION : 0.1
   VAR_INPUT
      mode : Bool;   // TRUE = select; FALSE = deselect
   END_VAR
   VAR_IN_OUT
      stations : "Stations";
   END_VAR
   VAR_TEMP
      btnCount : Int;
      i : Int;
      j : Int;
      selected : Bool;
      stnCount : Int;
   END_VAR
   VAR CONSTANT
      buttonCount : Int := 5;
   END_VAR
BEGIN
   REGION "COPY TO LOCAL"
       #btnCount := "ptsPerStn";
       #stnCount := "stnCount";
   END_REGION

   REGION "SELECT BUTTONS"
       FOR #i := 0 TO #stnCount DO

           REGION "SELCT ALL BUTTONS ON SELECTED STATION"
               #selected := #stations.me[#i].settings.selected;
               IF #selected THEN

                   REGION "LOOP THROUGH BUTTONS"
                       FOR #j := 0 TO #btnCount DO
                           #stations.me[#i].settings.btnSelection[#j] := #mode;
                       END_FOR;
                   END_REGION

               END_IF;
           END_REGION

       END_FOR;
   END_REGION
END_FUNCTION

FUNCTION "Animate Bool" : USInt   // FC9, SCL
{ S7_Optimized_Access := 'TRUE' }
VERSION : 0.1
   VAR_INPUT
      colorTrue : USInt;
      colorFalse : USInt;
      evalSignal : Bool;
   END_VAR
   VAR_TEMP
      animate : USInt;
   END_VAR
BEGIN
   REGION "FALSE COLOR"
       IF NOT #evalSignal THEN
           #animate := #colorFalse;
       END_IF;
   END_REGION

   REGION "TRUE COLOR"
       IF #evalSignal THEN
           #animate := #colorTrue;
       END_IF;
   END_REGION

   REGION "FUNCTION RETURN"
       #"Animate Bool" := #animate;
   END_REGION
END_FUNCTION

FUNCTION "WString to Time" : Time   // FC10, SCL
{ S7_Optimized_Access := 'TRUE' }
VERSION : 0.1
   VAR_INPUT
      WString : WString;
   END_VAR
   VAR_TEMP
      Count : UInt;
      "DInt Box" : DInt;
      "String Box" : WString [5];
      "Time Box" : Time;
      "WChar Array" : Array[0..4] of WChar;
   END_VAR
   VAR CONSTANT
      "ms/(10 hr)" : DInt := 36000000;
      "ms/hr" : DInt := 3600000;
      "ms/(10 min)" : DInt := 600000;
      "ms/min" : DInt := 60000;
      "ms/(10 sec)" : DInt := 10000;
      "ms/sec" : DInt := 1000;
   END_VAR
BEGIN
   REGION EXPLODE INPUT

       #"String Box" := #WString;
       IF #"String Box" = WSTRING#'' THEN
           #"String Box" := WSTRING#'00:00';
       END_IF;

       Strg_TO_Chars(Strg := #"String Box",
                     pChars := 0,
                     Cnt => #Count,
                     Chars := #"WChar Array");

   END_REGION

   REGION CONVERT ARRAY ELEMENTS TO TIME

       // 10S OF MINUTES
       #"DInt Box" := WCHAR_TO_DINT(IN := #"WChar Array"[0]) - 16#30;
       #"Time Box" := #"Time Box" + #"DInt Box" * #"ms/(10 min)";

       // MINUTES
       #"DInt Box" := WCHAR_TO_DINT(IN := #"WChar Array"[1]) - 16#30;
       #"Time Box" := #"Time Box" + #"DInt Box" * #"ms/min";

       // 10S OF SECONDS
       #"DInt Box" := WCHAR_TO_DINT(IN := #"WChar Array"[3]) - 16#30;
       #"Time Box" := #"Time Box" + #"DInt Box" * #"ms/(10 sec)";

       // SECONDS
       #"DInt Box" := WCHAR_TO_DINT(IN := #"WChar Array"[4]) - 16#30;
       #"Time Box" := #"Time Box" + #"DInt Box" * #"ms/sec";

   END_REGION


   REGION RETURN VALUE

       #"WString to Time" := #"Time Box";

   END_REGION
END_FUNCTION

FUNCTION "Get Part Call Row Number" : Int   // FC11, SCL
{ S7_Optimized_Access := 'TRUE' }
VERSION : 0.1
   VAR_IN_OUT
      partCall : "Part Call Screen";
   END_VAR
   VAR_TEMP
      hmiRows : Int;
      i : Int;
      selectedRow : Int;
   END_VAR
BEGIN
   REGION "GET NUMBER OF HMI ROWS"
       #hmiRows := "partReqHmiRowCount";
   END_REGION

   REGION "LOOP THROUGH HMI ROWS
       FOR #i := 0 TO #hmiRows DO

           REGION "FIND SELECTED ROW"
               IF #partCall.row[#i].pbSelection.actuate THEN
                   // selected row as int
                   #selectedRow := #i + 1;
                   EXIT;
               END_IF;
           END_REGION

       END_FOR;
   END_REGION

   REGION "RETURN ROW NUMBER"
       #"Get Part Call Row Number" := #selectedRow;
   END_REGION
END_FUNCTION

FUNCTION "Address to Station and Button" : Void   // FC12, SCL
{ S7_Optimized_Access := 'TRUE' }
VERSION : 0.1
   VAR_INPUT
      address : UInt;
   END_VAR
   VAR_OUTPUT
      station : UInt;
      button : UInt;
   END_VAR
BEGIN
   #station := #address / 10;
   #button := #address MOD 10;
END_FUNCTION

FUNCTION "WString Timer to Real" : Real   // FC13, SCL
{ S7_Optimized_Access := 'TRUE' }
VERSION : 0.1
   VAR_INPUT
      wstring : WString;
   END_VAR
   VAR CONSTANT
      msPerSec : Real := 1000.0;
   END_VAR
BEGIN
   #"WString Timer to Real" := DINT_TO_REAL(TIME_TO_DINT("WString to Time"(#wstring))) / #msPerSec;
END_FUNCTION

FUNCTION "Real to WString Timer" : WString   // FC14, SCL
{ S7_Optimized_Access := 'TRUE' }
VERSION : 0.1
   VAR_INPUT
      realVal : Real;
   END_VAR
   VAR CONSTANT
      msPerSec : Real := 1000.0;
   END_VAR
BEGIN
   #"Real to WString Timer" := "Time to WString"(DINT_TO_TIME(REAL_TO_DINT(#realVal * #msPerSec)));
END_FUNCTION

FUNCTION "Populate Dropzone IO Field" : WString   // FC15, SCL
{ S7_Optimized_Access := 'TRUE' }
VERSION : 0.1
   VAR_INPUT
      dzAsInt : USInt;
   END_VAR
BEGIN
   #"Populate Dropzone IO Field" := "Strip Sign"(USINT_TO_WSTRING(#dzAsInt));
END_FUNCTION

FUNCTION "Get Station Selection Number" : Void   // FC16, SCL
{ S7_Optimized_Access := 'TRUE' }
VERSION : 0.1
   VAR_INPUT
      next : Bool;   // 'next' or 'prev'
      prev : Bool;
      stations : "Stations";
   END_VAR
   VAR_IN_OUT
      selStnNumber : Int;
   END_VAR
   VAR_TEMP
      i : Int;
      stnCount : Int;
      stnSelected : Bool;
   END_VAR
BEGIN
   REGION "COPY TO LOCAL"
       #stnCount := "stnCount";
   END_REGION

   REGION "INITIALIZE INDEX"
       #i := #selStnNumber;
   END_REGION

   REGION "PREVIOUS MODE"

       REGION "DECREMENT"
           IF #prev THEN
               #i -= 1;
           END_IF;
       END_REGION

       REGION "LOW LIMIT ROLLOVER"
           IF #i < 0 THEN
               #i := #stnCount;
           END_IF;
       END_REGION

   END_REGION

   REGION "NEXT MODE"

       REGION "INCREMENT"
           IF #next THEN
               #i += 1;
           END_IF;
       END_REGION

       REGION "HIGH LIMIT ROLLOVER"
           IF #i > #stnCount THEN
               #i := 0;
           END_IF;
       END_REGION

   END_REGION

   REGION "COPY TO LOCAL"
       #stnSelected := #stations.me[#i].settings.selected;
   END_REGION

   REGION "FIND NEXT SELECTED STATION"
       WHILE NOT #stnSelected DO

           REGION "PREVIOUS MODE"

               REGION "DECREMENT"
                   IF #prev THEN
                       #i -= 1;
                   END_IF;
               END_REGION

               REGION "LOW LIMIT ROLLOVER"
                   IF #i < 0 THEN
                       #i := #stnCount;
                   END_IF;
               END_REGION

           END_REGION

           REGION "NEXT MODE"

               REGION "INCREMENT"
                   IF #next THEN
                       #i += 1;
                   END_IF;
               END_REGION

               REGION "HIGH LIMIT ROLLOVER"
                   IF #i > #stnCount THEN
                       #i := 0;
                   END_IF;
               END_REGION

           END_REGION

           REGION "SAVE WHILE CONDITION"
               #stnSelected := #stations.me[#i].settings.selected;
           END_REGION

       END_WHILE;
   END_REGION

   REGION "RETURN VALUE"
       #selStnNumber := #i;
   END_REGION
END_FUNCTION

FUNCTION "Populate Button Details" : Void   // FC17, SCL
{ S7_Optimized_Access := 'TRUE' }
VERSION : 0.1
   VAR_INPUT
      selStnNumber : Int;
      stations : "Stations";
   END_VAR
   VAR_IN_OUT
      settings : "Settings";
   END_VAR
   VAR_TEMP
      btnCount : Int;
      i : Int;
      partNumber : WString;
      pBtn : Int;
      timerWS : WString;
   END_VAR
BEGIN
   REGION "FOR EACH BUTTON"
       FOR #i := 0 TO "ptsPerStn" DO

           REGION "CALCULATE BUTTON POINTER"
               IF #i MOD 2 = 0 THEN
                   #pBtn := 7 - #i / 2;
               END_IF;
               IF #i MOD 2 <> 0 THEN
                   #pBtn := 3 - #i / 2;
               END_IF;
           END_REGION

           REGION "BUTTON LABEL"
               #settings.viewingStation.btns[#i].label.value := "Strip Sign"(INT_TO_WSTRING(#i + 1));
           END_REGION

           REGION "ALLOTTED TIME"
               #timerWS := "Real to WString Timer"(#stations.me[#selStnNumber].presetTime.allotted[#pBtn]);
               #settings.viewingStation.btns[#i].alloted.value := #timerWS;
           END_REGION

           REGION "CRITICAL TIME"
               #timerWS := "Real to WString Timer"(#stations.me[#selStnNumber].presetTime.critical[#pBtn]);
               #settings.viewingStation.btns[#i].critical.value := #timerWS;
           END_REGION

           REGION "PART NUMBER"
               #partNumber := #stations.me[#selStnNumber].partNumbers[#pBtn];
               #settings.viewingStation.btns[#i].partNumber.value := #partNumber;
           END_REGION

       END_FOR;
   END_REGION
END_FUNCTION

FUNCTION "Assign Station Parameters" : Void   // FC18, SCL
{ S7_Optimized_Access := 'TRUE' }
VERSION : 0.1
   VAR_IN_OUT
      settings : "Settings";
      stations : "Stations";
   END_VAR
   VAR_TEMP
      dzEntered : Bool;
      dzLabel : WString;
      i : Int;
      lineEntered : Bool;
      lineLabel : WString;
      stnCount : Int;
      stnSelected : Bool;
   END_VAR
BEGIN
   REGION "COPY TO LOCAL"    
       #dzEntered := #settings.viewingStation.dzData.inputFinished;
       #lineEntered := #settings.viewingStation.lineData.inputFinished;
       #stnCount := "stnCount";
   END_REGION

   REGION "ON PARAMETER ENTRY"
       IF #dzEntered OR #lineEntered THEN

           REGION "TURN OFF THE LIGHTS"
               #settings.viewingStation.dzData.inputFinished := FALSE;
               #settings.viewingStation.lineData.inputFinished := FALSE;
           END_REGION

           REGION "FOR EACH STATION"
               FOR #i := 0 TO #stnCount DO

                   REGION "COPY TO LOCAL"
                       #stnSelected := #stations.me[#i].settings.selected;
                   END_REGION

                   REGION "ON SELECTED STATION"
                       IF #stnSelected THEN

                           REGION "ON DROP ZONE INPUT"
                               IF #dzEntered THEN

                                   REGION "GET FROM HMI"
                                       #dzLabel := #settings.viewingStation.dzData.value;
                                   END_REGION

                                   REGION "WRITE TO STATION PARAMETER"
                                       #stations.me[#i].dropZone := WSTRING_TO_USINT(#dzLabel);
                                   END_REGION

                               END_IF;
                           END_REGION

                           REGION "ON LINE LABEL INPUT"
                               IF #lineEntered THEN

                                   REGION "GET FROM HMI"
                                       #lineLabel := #settings.viewingStation.lineData.value;
                                   END_REGION

                                   REGION "WRITE TO STATION PARAMETER"
                                       #stations.me[#i].line := #lineLabel;
                                   END_REGION

                               END_IF;
                           END_REGION

                       END_IF;
                   END_REGION

               END_FOR;
           END_REGION

       END_IF;
   END_REGION
END_FUNCTION

FUNCTION "Animate Button Details" : Void   // FC19, SCL
{ S7_Optimized_Access := 'TRUE' }
VERSION : 0.1
   VAR_INPUT
      stations : "Stations";
   END_VAR
   VAR_IN_OUT
      settings : "Settings";
   END_VAR
   VAR_TEMP
      animate : USInt;
      btnCount : Int;
      btnSelected : Bool;
      deselected : USInt;
      i : Int;
      invisible : USInt;
      pBtn : Int;
      selected : USInt;
      selStnCount : Int;
      selStnNumber : Int;
   END_VAR
BEGIN
   REGION "COPY TO LOCAL"
       #btnCount := "ptsPerStn";
       #deselected := "BgGray";
       #invisible := "invisible";
       #selected := "BgLTe";
       #selStnCount := #settings.#stations.selCount;
       #selStnNumber := #settings.stations.selNumber;
   END_REGION

   REGION "ENABLE"
       IF #selStnCount >= 1 THEN

           REGION "SHOW BUTTON DETAILS"
               #animate := #deselected;
           END_REGION

       END_IF;
   END_REGION

   REGION "DISABLE"
       IF #selStnCount = 0 THEN

           REGION "HIDE BUTTON DETAILS"
               #animate := #invisible;
           END_REGION

       END_IF;
   END_REGION

   REGION "APPLY ANIMATION"
       FOR #i := 0 TO #btnCount DO

           REGION "CALCULATE BUTTON POINTER"
               #pBtn := "Pointer Calc: Button Details"(#i);
           END_REGION

           REGION "WHILE Station SELECTED"
               IF #selStnCount <> 0 THEN

                   REGION "COPY TO LOCAL"
                       #btnSelected := #stations.me[#selStnNumber].settings.btnSelection[#pBtn];
                   END_REGION

                   REGION "ANIMATE BUTTON SELECTION

                       REGION "SELECTED"
                           IF #btnSelected THEN
                               #animate := #selected;
                           END_IF;
                       END_REGION

                       REGION "NOT SELECTED"
                           IF NOT #btnSelected THEN
                               #animate := #deselected;
                           END_IF;
                       END_REGION

                   END_REGION

               END_IF;
           END_REGION


           REGION "SEND TO HMI"
               #settings.viewingStation.btns[#i].label.animate := #animate;
               #settings.viewingStation.btns[#i].alloted.animate := #animate;
               #settings.viewingStation.btns[#i].critical.animate := #animate;
               #settings.viewingStation.btns[#i].partNumber.animate := #animate;
           END_REGION

       END_FOR;
   END_REGION
END_FUNCTION

FUNCTION "Populate Station Name" : WString   // FC20, SCL
{ S7_Optimized_Access := 'TRUE' }
VERSION : 0.1
   VAR_INPUT
      line : WString;
      dropZone : USInt;
   END_VAR
BEGIN
   #"Populate Station Name" := CONCAT_WSTRING(IN1 := #line,
                                              IN2 := wstring#' ',
                                              IN3 := "Strip Sign"(USINT_TO_WSTRING(#dropZone)));
END_FUNCTION

FUNCTION "Pointer Calc: Button Details" : Int   // FC21, SCL
{ S7_Optimized_Access := 'TRUE' }
VERSION : 0.1
   VAR_INPUT
      index : Int;
   END_VAR
   VAR_TEMP
      val : Int;
   END_VAR
BEGIN
   IF #index MOD 2 = 0 THEN
       #val := 7 - #index / 2;
   END_IF;

   IF #index MOD 2 <> 0 THEN
       #val := 3 - #index / 2;
   END_IF;

   #"Pointer Calc: Button Details" := #val;
END_FUNCTION

FUNCTION "Buffer Part Req Log Row: Generate" : "Part Req Log Row"   // FC22, SCL
{ S7_Optimized_Access := 'TRUE' }
VERSION : 0.1
   VAR_INPUT
      address : Int;
      "type" : Int;
   END_VAR
   VAR_TEMP
      retVal : Int;
   END_VAR
BEGIN
   REGION "ADDRESS"
       #"Buffer Part Req Log Row: Generate".address := #address;
   END_REGION

   REGION "REQUEST TYPE"
       #"Buffer Part Req Log Row: Generate".reqType := #type;
   END_REGION

   REGION "TIME STAMP"
       #retVal := RD_SYS_T(#"Buffer Part Req Log Row: Generate".timeStamp);
   END_REGION
END_FUNCTION

FUNCTION "Sim to Global" : Void   // FC23, SCL
{ S7_Optimized_Access := 'TRUE' }
VERSION : 0.1
   VAR_INPUT
      simStations : "Simulated Stations";
   END_VAR
   VAR_IN_OUT
      stations : "Stations";
   END_VAR
   VAR_TEMP
      btnCount : Int;
      firstStn : Int;
      i : Int;
      j : Int;
      pSim : Int;
      pStn : Int;
      simKP8Count : Int;
      stnCount : Int;
   END_VAR
BEGIN
   REGION "COPY TO LOCAL"
       #btnCount := "ptsPerStn";
       #firstStn := #simStations.firstStn;
       #simKP8Count := "simKP8Count";
       #stnCount := "stnCount";
   END_REGION

   REGION "FOR EACH STATION"
       FOR #i := 0 TO #simKP8Count DO

           REGION "CALCULATE POINTER"
               #pStn := #i + #firstStn;
               #pSim := #i;
           END_REGION

           REGION "UPPER LIMIT ROLL OVER"
               IF #pStn > #stnCount THEN
                   #pStn := #firstStn + #i - #stnCount - 1;
               END_IF;
           END_REGION

           REGION "COPY SIMULATED PRESSES"
               #stations.me[#pStn].kp8In := #simStations.me[#pSim].btn.actuate;
           END_REGION

       END_FOR;
   END_REGION
END_FUNCTION

FUNCTION "HSS: Template" : Void   // FC24, SCL
{ S7_Optimized_Access := 'TRUE' }
VERSION : 0.1
   VAR_INPUT
      menuLibrary : "Recipe: Library";
      menuSelector : Int;
   END_VAR
   VAR_IN_OUT
      tmplt : "HSS: Template Screen";
   END_VAR
   VAR_TEMP
      i : Int;
   END_VAR
BEGIN
   #tmplt.animate[0] := "BgGray";
   #tmplt.text[0] := "Word Wrap"(stringIn := #menuLibrary.wip[#menuSelector],
                                 maxLength := 22);
END_FUNCTION

FUNCTION "Pointer Calc: KP8 Labels" : Int   // FC25, SCL
{ S7_Optimized_Access := 'TRUE' }
VERSION : 0.1
   VAR_INPUT
      index : Int;
   END_VAR
   VAR_TEMP
      val : Int;
   END_VAR
BEGIN
   IF #index >= 4 THEN
       #val := 7 - (#index - 4) * 2;
   END_IF;

   IF #index <= 3 THEN
       #val := 8 - #index * 2;
   END_IF;

   #"Pointer Calc: KP8 Labels" := #val;
END_FUNCTION

FUNCTION "KP8 Color to Sim Animation" : USInt   // FC26, SCL
{ S7_Optimized_Access := 'TRUE' }
VERSION : 0.1
   VAR_INPUT
      kp8Color : DWord;
      btnNumber : Int;
   END_VAR
   VAR_TEMP
      animate : USInt;
      blue : USInt;
      colorDWord : DWord;
      colorInt : DInt;
      green : USInt;
      off : USInt;
      red : USInt;
      white : USInt;
      yellow : USInt;
   END_VAR
   VAR CONSTANT
      blueMask : DInt := 16#0000_0100;
      btnMask : DInt := 16#0101_0100;
      greenMask : DInt := 16#0001_0000;
      offMask : DInt := 16#0000_0000;
      redMask : DInt := 16#0100_0000;
      whiteMask : DInt := 16#0101_0100;
      yellowMask : DInt := 16#0101_0000;
   END_VAR
BEGIN
   REGION "COPY TO LOCAL"
       #blue := "BgLBl";
       #green := "BgLGr";
       #off := "BgGray";
       #red := "BgLRd";
       #white := "BgWh";
       #yellow := "BgLYe";
   END_REGION

   REGION "ISOLATE BUTTON COLOR"
       #colorDWord := SHR_DWORD(IN := #kp8Color,N := INT_TO_ULINT(#btnNumber));
       #colorDWord := #colorDWord AND #btnMask;
       #colorInt := DWORD_TO_DINT(#colorDWord);
   END_REGION

   REGION "DETERMINE ANIMATION"
       CASE #colorInt OF
           #blueMask:
               #animate := #blue;
           #greenMask:
               #animate := #green;
           #redMask:
               #animate := #red;
           #whiteMask:
               #animate := #white;
           #yellowMask:
               #animate := #yellow;
           ELSE
               #animate := #off;
       END_CASE;
   END_REGION

   REGION "RETURN VALUE"
       #"KP8 Color to Sim Animation" := #animate;
   END_REGION
END_FUNCTION

FUNCTION "Initialize Recipe Select Screens" : Void   // FC27, SCL
{ S7_Optimized_Access := 'TRUE' }
VERSION : 0.1
   VAR_INPUT
      libs : "Recipe: Libraries";
   END_VAR
   VAR_IN_OUT
      slctScreen : Array[0.."hmiStnCount"] of "HSS: Compressed";
   END_VAR
   VAR_TEMP
      j : Int;
      maxRows : Int;
      i : Int;
   END_VAR
   VAR CONSTANT
      visRows : Int := 6;
   END_VAR
BEGIN
   REGION "LABELS"
       FOR #i := 25 TO 29 DO
           #maxRows := #libs.stations[#i].size;
           IF #maxRows > 0 THEN
               FOR #j := 0 TO #visRows - 1 DO
                   IF #j <= 5 THEN
                       "Recipe Nav Button"(visRows := #visRows,
                                           actuate := FALSE,
                                           maxRows := #maxRows,
                                           btnNum := #j,
                                           recipeSelectScreen := #slctScreen[#i - 25].scrnSlctMn);
                   END_IF;
                   "Recipe Select Button"(visRows := #visRows,
                                          rowNum := #j,
                                          lib := #libs.stations[25],
                                          actuate := FALSE,
                                          maxRows := #maxRows,
                                          btnNum := #j,
                                          recipeSelectScreen := #slctScreen[#i - 25].scrnSlctMn);
               END_FOR;
           END_IF;
       END_FOR;
   END_REGION
END_FUNCTION

FUNCTION "Word Wrap" : WString   // FC28, SCL
{ S7_Optimized_Access := 'TRUE' }
VERSION : 0.1
   VAR_INPUT
      stringIn : WString;
      maxLength : Int;
   END_VAR
   VAR_TEMP
      length : Int;
      charBox : Array[0.."lStringLen"] of WChar;
      stringBox : Array[0.."lStringLen"] of WString["lStringLen"];
      count : UInt;
      status : Int;
      i : Int;
      pStringBox : Int;
      output : WString;
      savedOutput : WString;
      lineBox : Array[0..10] of WString["lStringLen"];
      pLineBox : Int;
      lengthTest : WString;
   END_VAR
   VAR CONSTANT
      space : WString := WSTRING#' ';
      blank : WString;
      lineBreak : WString := WSTRING#'$L';
   END_VAR
BEGIN
   #length := LEN(#stringIn);

   IF #length <= #maxLength THEN
       #output := #stringIn;
   END_IF;

   IF #length > #maxLength THEN

       Strg_TO_Chars(
                     Strg := #stringIn,
                     pChars := 0,
                     Cnt => #count,
                     Chars := #charBox
       );

       FOR #i := 0 TO "lStringLen" DO

           IF #charBox[#i] = #space THEN
               IF #charBox[#i + 1] = #space THEN
                   EXIT;
               END_IF;
           END_IF;

           IF #i = 0 THEN
               #stringBox[#pStringBox] := #charBox[#i];
           END_IF;

           IF #i >= 1 THEN
               #stringBox[#pStringBox] := CONCAT_WSTRING(IN1 := #stringBox[#pStringBox],
                                                         IN2 := #charBox[#i]);
           END_IF;

           IF #charBox[#i] = #space THEN
               #stringBox[#pStringBox] := "Trim"(#stringBox[#pStringBox]);
               #pStringBox := #pStringBox + 1;
           END_IF;

           IF #charBox[#i] = #lineBreak THEN
               #stringBox[#pStringBox] := LEFT(IN := #stringBox[#pStringBox],
                                               L := LEN(#stringBox[#pStringBox]) - 1);
               #pStringBox := #pStringBox + 1;
               #stringBox[#pStringBox] := #lineBreak;
               #pStringBox := #pStringBox + 1;
           END_IF;

       END_FOR;


       FOR #i := 0 TO "lStringLen" DO

           IF #stringBox[#i] = #blank THEN
               IF #stringBox[#i + 1] = #blank THEN
                   #lineBox[#pLineBox] := "Trim"(#lineBox[#pLineBox]);
                   EXIT;
               END_IF;
           END_IF;

           IF #stringBox[#i] = #lineBreak THEN
               #lineBox[#pLineBox] := "Trim"(#lineBox[#pLineBox]);
               #pLineBox := #pLineBox + 1;
               #lineBox[#pLineBox] := #lineBreak;
               #pLineBox := #pLineBox + 1;
           END_IF;


           IF #stringBox[#i] <> #lineBreak THEN

               IF #i = 0 THEN
                   #lengthTest := #stringBox[#i];
               END_IF;

               IF #i >= 1 THEN
                   #lengthTest := CONCAT_WSTRING(IN1 := #lineBox[#pLineBox],
                                                 IN2 := #space,
                                                 IN3 := #stringBox[#i]);
               END_IF;

               IF LEN(#lengthTest) <= #maxLength THEN
                   #lineBox[#pLineBox] := #lengthTest;
               END_IF;

               IF LEN(#lengthTest) > #maxLength THEN
                   #lineBox[#pLineBox] := "Trim"(#lineBox[#pLineBox]);
                   #lineBox[#pLineBox] := "Trim"(#lineBox[#pLineBox]);
                   #pLineBox := #pLineBox + 1;
                   #lineBox[#pLineBox] := #stringBox[#i];
               END_IF;
           END_IF;

       END_FOR;

       FOR #i := 0 TO 10 DO

           IF #lineBox[#i] = #space OR #lineBox[#i] = WString#'' THEN
               EXIT;
           END_IF;
           IF #i = 0 THEN
               #output := #lineBox[#i];
           END_IF;
           IF #i >= 1 THEN
               IF #lineBox[#i] = #lineBreak THEN
                   #output := #output;
               END_IF;
               IF #lineBox[#i] <> #lineBreak THEN
                   #output := CONCAT_WSTRING(IN1 := #output,
                                             IN2 := #lineBreak,
                                             IN3 := #lineBox[#i]);
               END_IF;
           END_IF;

       END_FOR;

       #output := "Trim"(#output);

   END_IF;

   #"Word Wrap" := #output;
END_FUNCTION

FUNCTION "Trim" : WString   // FC29, SCL
{ S7_Optimized_Access := 'TRUE' }
VERSION : 0.1
   VAR_INPUT
      stringIn : WString;
   END_VAR
   VAR_TEMP
      output : WString;
   END_VAR
   VAR CONSTANT
      space : WString := WSTRING#' ';
   END_VAR
BEGIN
   #output := #stringIn;
   IF LEFT(IN := #output, L := 1) = #space THEN
       #output := RIGHT(IN := #output, L := LEN(#output) - 1);
   END_IF;
   IF RIGHT(IN := #output, L := 1) = #space THEN
       #output := LEFT(IN := #output, L := LEN(#output) - 1);
   END_IF;
   #Trim := #output;
END_FUNCTION

FUNCTION "Get Recipes Per Station" : Void   // FC30, SCL
{ S7_Optimized_Access := 'TRUE' }
VERSION : 0.1
   VAR_INPUT
      libs : "Recipe: Libraries";
   END_VAR
   VAR_TEMP
      i : Int;
      j : Int;
      thisEntry : WString;
      size : Int;
   END_VAR
   VAR CONSTANT
      blank : WString;
   END_VAR
BEGIN
   FOR #i := 0 TO "stnCount" DO
       #size := 0;
       FOR #j := 0 TO "menuCntPerStn" DO
           #thisEntry := #libs.stations[#i].wip[#j];
           IF #thisEntry <> #blank THEN
               #size += 1;
           END_IF;
       END_FOR;
       "Recipe Libraries".me.stations[#i].size := #size;
   END_FOR;
END_FUNCTION

FUNCTION "Recipe Select Button" : Void   // FC31, SCL
{ S7_Optimized_Access := 'TRUE' }
VERSION : 0.1
   VAR_INPUT
      visRows : Int;
      rowNum : Int;
      lib : "Recipe: Library";
      actuate : Bool;
      maxRows : Int;
      btnNum : Int;
   END_VAR
   VAR_IN_OUT
      recipeSelectScreen : "HSS: Menu Selection Screen";
   END_VAR
   VAR_TEMP
      eval : "HSS: Menu Selection Screen";
      pRowVisLbl : Int;
      pRowInvisLbl : Int;
      pRowTxt : Int;
      pRecipeTxt : Int;
      maxLen : Int;
   END_VAR
BEGIN
   REGION "COPY TO LOCAL"
       #eval := #recipeSelectScreen;
   END_REGION


   REGION "NARROW"
       IF #maxRows > #visRows THEN
           #pRowVisLbl := #btnNum + #visRows;
           #pRowInvisLbl := #btnNum + (3 * #visRows);
           #maxLen := 22;
       END_IF;
   END_REGION


   REGION "WIDE"
       IF #maxRows <= #visRows THEN
           #pRowVisLbl := #btnNum + (3 * #visRows);
           #pRowInvisLbl := #btnNum + #visRows + 1;
           #maxLen := 28;
       END_IF;
   END_REGION


   REGION "ROW COUNT INDEPENDENT"
       #pRowTxt := (#btnNum * 2) + #visRows;
       #pRecipeTxt := #pRowTxt + 1;
   END_REGION


   REGION "DRAW"
       IF #btnNum < #maxRows THEN
           #eval.animate[#pRowVisLbl] := "BgGray";
       END_IF;
       IF #btnNum >= #maxRows THEN
           #eval.animate[#pRowVisLbl] := "invisible";
       END_IF;
       #eval.animate[#pRowInvisLbl] := "invisible";
       #eval.txt[#pRowTxt] := "Strip Sign"(DINT_TO_WSTRING(#rowNum));
       #eval.txt[#pRecipeTxt] := "Word Wrap"(stringIn := #lib.wip[#rowNum],
                                             maxLength := #maxLen);
   END_REGION

   REGION "ACTUATION ANIMATION"
       IF #actuate THEN
           #eval.animate[#pRowVisLbl] := "BgLTe";
       END_IF;
   END_REGION


   REGION "COPY TO GLOBAL"
       #recipeSelectScreen := #eval;
   END_REGION
END_FUNCTION

FUNCTION "Recipe Nav Button" : Void   // FC32, SCL
{ S7_Optimized_Access := 'TRUE' }
VERSION : 0.1
   VAR_INPUT
      visRows : Int;
      actuate : Bool;
      maxRows : Int;
      btnNum : Int;
   END_VAR
   VAR_IN_OUT
      recipeSelectScreen : "HSS: Menu Selection Screen";
   END_VAR
   VAR_TEMP
      eval : "HSS: Menu Selection Screen";
      color : Int;
   END_VAR
BEGIN
   REGION "COPY TO LOCAL"
       #eval := #recipeSelectScreen;
   END_REGION


   REGION "NARROW"
       IF #maxRows > #visRows THEN
           #color := "BgGray";
       END_IF;
   END_REGION


   REGION "WIDE"
       IF #maxRows <= #visRows THEN
           #color := "invisible";
       END_IF;
   END_REGION


   REGION "ROW COUNT INDEPENDENT"
       IF #actuate THEN
           #color := "BgLTe";
       END_IF;
   END_REGION


   REGION "DRAW"
       #eval.animate[#btnNum] := #color;
   END_REGION


   REGION "COPY TO GLOBAL"
       #recipeSelectScreen := #eval;
   END_REGION
END_FUNCTION

FUNCTION "Initialize Part Select Screens" : Void   // FC33, SCL
{ S7_Optimized_Access := 'TRUE' }
VERSION : 0.1
   VAR_INPUT
      libs : "Recipe: Libraries";
      recipeNum : Int;
      stations : "Stations";
   END_VAR
   VAR_IN_OUT
      slctScreen : Array[0.."hmiStnCount"] of "HSS: Compressed";
   END_VAR
   VAR_TEMP
      i : Int;
      j : Int;
   END_VAR
BEGIN
   REGION "LABELS"
       FOR #i := 25 TO 29 DO
           FOR #j := 0 TO "ptsPerStn" DO
               "Part Select Button"(recipeNum := #recipeNum,
                                    lib := #libs.stations[#i],
                                    actuate := FALSE,
                                    btnNum := #j,
                                    stn := #stations.me[#i],
                                    partSelectScreen := #slctScreen[#i - 25].scrnSlctPrt);
           END_FOR;
       END_FOR;
   END_REGION
END_FUNCTION

FUNCTION "Part Select Button" : Void   // FC34, SCL
{ S7_Optimized_Access := 'TRUE' }
VERSION : 0.1
   VAR_INPUT
      recipeNum : Int;
      lib : "Recipe: Library";
      actuate : Bool;
      btnNum : Int;
      stn : "Station";
   END_VAR
   VAR_IN_OUT
      partSelectScreen : "HSS: Part Selection Screen";
   END_VAR
   VAR_TEMP
      eval : "HSS: Part Selection Screen";
      i : Int;
      target : Int;
   END_VAR
   VAR CONSTANT
      blank : WString;
      anDefault : USInt := 0;
      anRequested : USInt := 1;
      anSolidRed : USInt := 2;
      anFlashRed : USInt := 3;
      anPartOrdered : USInt := 4;
   END_VAR
BEGIN
   REGION "COPY TO LOCAL"
       #eval := #partSelectScreen;
   END_REGION


   REGION "DRAW NEEDED BUTTONS"
       IF #stn.partNumbers[#btnNum] = #blank THEN
           #eval.animate[#btnNum] := "invisible";
       END_IF;
       IF #stn.partNumbers[#btnNum] <> #blank THEN
           CASE #stn.animations[#btnNum] OF
               #anDefault:
                   #eval.animate[#btnNum] := "BgLGr";
               #anRequested:
                   #eval.animate[#btnNum] := "BgDYe";
               #anSolidRed:
                   #eval.animate[#btnNum] := "BgDRd";
               #anFlashRed:
                   #eval.animate[#btnNum] := "FlDrd";
               #anPartOrdered:
                   #eval.animate[#btnNum] := "BgDBl";
               ELSE:
                   ;
           END_CASE;
       END_IF;
   END_REGION


   REGION "ACTUATION ANIMATION"
       IF #actuate THEN
           #eval.animate[#btnNum] := "BgLTe";
       END_IF;
   END_REGION


   REGION "PART NUMBER"
       #eval.txt[#btnNum] :=#stn.partNumbers[#btnNum];
   END_REGION


   REGION "COPY TO GLOBAL"
       #partSelectScreen := #eval;
   END_REGION
END_FUNCTION

FUNCTION "LRUD KP8 Remap" : Int   // FC35, SCL
{ S7_Optimized_Access := 'TRUE' }
VERSION : 0.1
   VAR_INPUT
      btnNum : Int;
      mode : Int;   // 1 = KP8; 2 = KTP700
   END_VAR
   VAR_TEMP
      output : Int;
   END_VAR
   VAR CONSTANT
      kp8 : Int := 1;
      ktp700 : Int := 2;
   END_VAR
BEGIN
   IF #btnNum >= 4 THEN
       #output := (7 - #btnNum) * 2;
   END_IF;

   IF #btnNum <= 3 THEN
       #output := (3 - #btnNum) * 2 + 1;
   END_IF;

   #"LRUD KP8 Remap" := #output;
END_FUNCTION

FUNCTION "Retain Button States" : Void   // FC36, SCL
{ S7_Optimized_Access := 'TRUE' }
VERSION : 0.1
   VAR_INPUT
      firstScan : Bool;
      initialize : Bool;
   END_VAR
   VAR_TEMP
      i : Int;
      j : Int;
   END_VAR
BEGIN
   FOR #i := 0 TO "stnCount" DO
           FOR #j := 0 TO "ptsPerStn" DO
               IF #firstScan THEN
                   "EMP IDB".instKP8Drvs[#i].btnStateArrayInt[#j] :=
                   "EMP IDB".stations.me[#i].btnStates[#j];
               END_IF;
               IF #initialize THEN
                   "EMP IDB".instKP8Drvs[#i].btnStateArrayInt[#j] := FALSE;
                   "EMP IDB".stations.me[#i].btnStates[#j] := FALSE;
               END_IF;
           END_FOR;
   END_FOR;
END_FUNCTION

ORGANIZATION_BLOCK "Main"   // OB1, LAD, ProgramCycle
TITLE = "Main Program Sweep (Cycle)"
{ S7_Optimized_Access := 'TRUE' }
VERSION : 0.1
   VAR_INPUT
      Initial_Call : Bool;   // Initial call of this OB
      Remanence : Bool;   // =True, if remanent data are available
   END_VAR
BEGIN

REGION Network 1
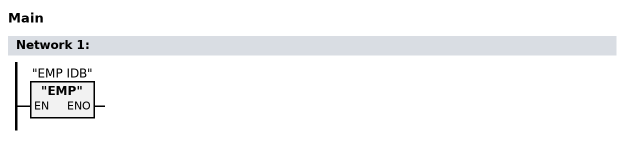
   RUNG wire#powerrail
      "EMP IDB"()
   END_RUNG
   // the same network as SCL:
   "EMP IDB"();   // "EMP"
END_REGION
END_ORGANIZATION_BLOCK

ORGANIZATION_BLOCK "Rack or station failure"   // OB86, LAD, RackStationFailure
{ S7_Optimized_Access := 'TRUE' }
VERSION : 0.1
   VAR_INPUT
      LADDR : Hw_Device;   // Hardware identifier
      Event_Class : Byte;   // Event class
      Fault_ID : Byte;   // Fault identifier
   END_VAR
BEGIN
END_ORGANIZATION_BLOCK

ORGANIZATION_BLOCK "Startup"   // OB100, LAD, Startup
TITLE = "Complete Restart"
{ S7_Optimized_Access := 'TRUE' }
VERSION : 0.1
// //============================================================================
// //SIEMENS AG
// //(c)Copyright 2017 All Rights Reserved
// //-----------------------------------------------------------------------------
// //Library: -
// //Tested with: S7-1516-3 PN/DP FW 2.5
// //Engineering: TIA Portal V15
// //Restrictions: -
// //Requirements: -
// //Functionality: Startup OB for Diagnostics
// //-----------------------------------------------------------------------------
// //Change log table:
// //Version  Date              Expert in charge                               Changes applied
// //01.00.00 25.04.2017 Siemens Industry Online Support First released version
// //============================================================================
   VAR_INPUT
      LostRetentive : Bool;   // True if retentive data are lost
      LostRTC : Bool;   // True if date and time are lost
   END_VAR
   VAR_TEMP
      index : Int;
   END_VAR
BEGIN

REGION Network 1: Set start user diagnostic
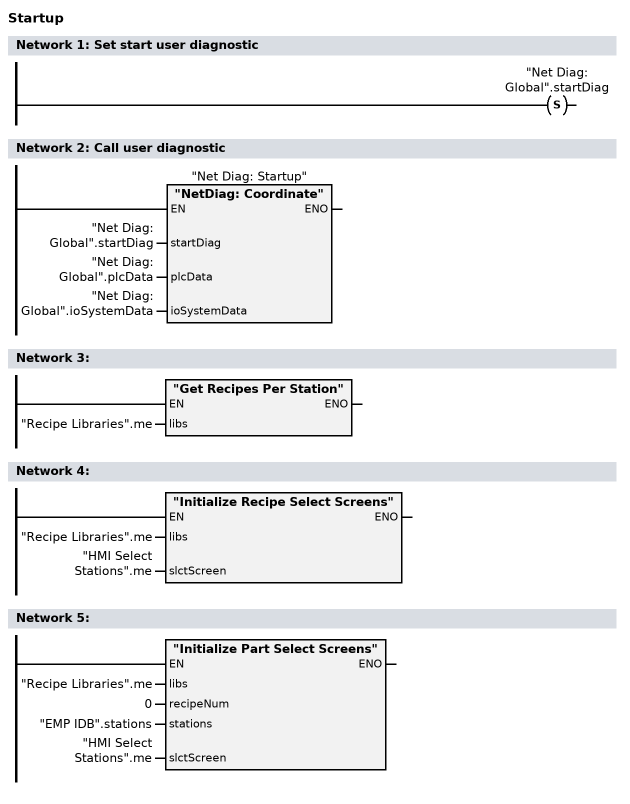
   RUNG wire#powerrail
      S_Coil( "Net Diag: Global".startDiag )
   END_RUNG
   // the same network as SCL:
   "Net Diag: Global".startDiag := TRUE;
END_REGION

REGION Network 2: Call user diagnostic
   RUNG wire#powerrail
      "Net Diag: Startup"(startDiag := "Net Diag: Global".startDiag, plcData := "Net Diag: Global".plcData, ioSystemData := "Net Diag: Global".ioSystemData)
   END_RUNG
   // the same network as SCL:
   "Net Diag: Startup"(startDiag := "Net Diag: Global".startDiag,   // "NetDiag: Coordinate"
                       plcData := "Net Diag: Global".plcData,
                       ioSystemData := "Net Diag: Global".ioSystemData);
END_REGION

REGION Network 3
   RUNG wire#powerrail
      "Get Recipes Per Station"(libs := "Recipe Libraries".me)
   END_RUNG
   // the same network as SCL:
   "Get Recipes Per Station"(libs := "Recipe Libraries".me);
END_REGION

REGION Network 4
   RUNG wire#powerrail
      "Initialize Recipe Select Screens"(libs := "Recipe Libraries".me, slctScreen := "HMI Select Stations".me)
   END_RUNG
   // the same network as SCL:
   "Initialize Recipe Select Screens"(libs := "Recipe Libraries".me, slctScreen := "HMI Select Stations".me);
END_REGION

REGION Network 5
   RUNG wire#powerrail
      "Initialize Part Select Screens"(libs := "Recipe Libraries".me, recipeNum := 0, stations := "EMP IDB".stations, slctScreen := "HMI Select Stations".me)
   END_RUNG
   // the same network as SCL:
   "Initialize Part Select Screens"(libs := "Recipe Libraries".me,
                           recipeNum := 0,
                           stations := "EMP IDB".stations,
                           slctScreen := "HMI Select Stations".me);
END_REGION
END_ORGANIZATION_BLOCK

ORGANIZATION_BLOCK "Programming error"   // OB121, LAD, ProgrammingError
{ S7_Optimized_Access := 'TRUE' }
VERSION : 0.1
   VAR_INPUT
      BlockNr : UInt;   // Number of causing block
      Reaction : USInt;   // 0:ignore, 1:substitute, 2:skip
      Fault_ID : Byte;   // Fault identifier
      BlockType : USInt;   // 16#01:OB, 16#02:FC, 16#03:FB, 16#04:SFC, 16#05:SFB, 16#06:DB: Type of block causing the error
      Area : USInt;   // Area where the error occured
      DBNr : DB_ANY;   // DB number if Area = DB or DI
      Csg_OBNr : OB_Any;   // Number of OB causing the error
      Csg_Prio : USInt;   // Priority of OB causing the error
      Width : USInt;   // 0:bit, 1:byte, 2:word, 3:dword, 4:lword
   END_VAR
BEGIN
END_ORGANIZATION_BLOCK

ORGANIZATION_BLOCK "IO access error"   // OB122, LAD, IOAccessError
{ S7_Optimized_Access := 'TRUE' }
VERSION : 0.1
   VAR_INPUT
      BlockNr : UInt;   // Number of causing block
      Reaction : USInt;   // 0:ignore, 1:substitute, 2:skip
      Fault_ID : Byte;   // 16#42:reading, 16#43:writing
      BlockType : USInt;   // 16#01:OB, 16#02:FC, 16#03:FB, 16#04:SFC, 16#05:SFB, 16#06:DB: Type of block causing the error
      Area : USInt;   // 16#81:I, 16#82:Q: IO area where the IOaccess error occured
      DBNr : DB_ANY;   // Reserved for system
      Csg_OBNr : OB_Any;   // Number of OB causing the error
      Csg_Prio : USInt;   // Priority of OB causing the error
      Width : USInt;   // 0:bit, 1:byte, 2:word, 3:dword, 4:lword
   END_VAR
BEGIN
END_ORGANIZATION_BLOCK

// ===== library types =====

TYPE "Table Row Data"
VERSION : 0.1
   STRUCT
      address : UInt;
      ordered : Bool;
      pbSelection : Struct
         actuate : Bool;
         animate : USInt;
      END_STRUCT;
      rtBackground : Struct
         animate : USInt;
      END_STRUCT;
      tfDropZone : Struct
         animate : USInt;
         value : WString[20];
      END_STRUCT;
      tfLine : Struct
         animate : USInt;
         value : WString[20];
      END_STRUCT;
      tfPartNumber : Struct
         animateDL : USInt;
         animateSL : USInt;
         value : WString[40];
      END_STRUCT;
      tfTime : Struct
         animate : USInt;
         value : WString[20];
      END_STRUCT;
   END_STRUCT;
END_TYPE

TYPE "Station Assignment: Button Details Data"
VERSION : 0.1
   STRUCT
      alloted : Struct
         animate : USInt;
         value : WString[10];
      END_STRUCT;
      critical : Struct
         animate : USInt;
         value : WString[10];
      END_STRUCT;
      label : Struct
         animate : USInt;
         value : WString[2];
      END_STRUCT;
      partNumber : Struct
         animate : USInt;
         value : WString[40];
      END_STRUCT;
      select : Struct
         actuate : Bool;
         animate : USInt;
      END_STRUCT;
   END_STRUCT;
END_TYPE